TYPE "digital_inputs"
VERSION : 0.1
   STRUCT
       OtwAKPiA : Bool;    // Otawrcie szafy AKPiA
    "Czujn_Zal>0.2m" : Bool;    // Obecność w komorze AKPiA
    "Czujn_Zal>1m" : Bool;    // Obecność w komorze podziemnej
    Zasilanie : Bool;    // Obecność w komorze naziemnej
    ObcKom : Bool;    // Zalanie komory > 0.2m
    ZasilDRC : Bool;    // Zasilanie czujnika ruchu CZ1
    ZasilPompOdw : Bool;    // Zasilanie kontakorna otwarcia drzwi
    ZasilPlywZalania : Bool;    // Zasilanie czujnika ruchu CZ2
    ZasilCzujnRuchu : Bool;    // Zasilanie czujnika ruchu CZ3
    ZasilKontaktDrzwi : Bool;    // Zasilanie pływaka komory podziemnej
END_STRUCT;

END_TYPE
TYPE "digital_outputs"
VERSION : 0.1
   STRUCT
       "void" : Bool ;
   END_STRUCT;
END_TYPE
   TYPE "analog_outputs"
VERSION : 0.1
   STRUCT
       "void" : Bool ;
   END_STRUCT;
END_TYPE
   TYPE "analog_inputs"
VERSION : 0.1
   STRUCT
       FT01_Przeplyw : Int;    // Przepływ
    TTs_TempSzafy : Int;    // Temperatura szafy
    TTz_TempZewn : Int;    // Temperatura zawenętrzna
    PT07_CisnZasil_WRZ6 : Int;    // Ciśnienie w kierunku WRZ6
    PT08_CisnPowr_WRZ6 : Int;    // Ciśnienie powrotu z WRZ6
    TTk_TempKom : Int;    // Temperatura w komorze podziemnej
    PT01_CisnZasil_PLN1 : Int;    // Ciśnienie zasilania z PLN1
    PT02_CisnPowr_PLN1 : Int;    // Ciśnienie powrotu w kierunku PLN1
    PT03_CisnZasil_Bypass : Int;    // Ciśnienie zasilania Bypass
    PT04_CisnPowr_Bypass : Int;    // Ciśnienie powrotu Bypass
    PT05_CisnZasil_PLN12 : Int;    // Ciśnienie zasilania w kierunku PLN12
    PT06_CisnPowr_PLN12 : Int;    // Ciśnienie powrotu z PLN12
    TT01_TempZasil_PLN1 : Int;    // Temperatura zasliania z PLN1
    TT02_TempPowr_PLN1 : Int;    // Temperatura powrotu w kierunku PLN1
    TT04_TempPowr_WRZ6 : Int;    // Temperatura powrotu z WRZ6
    TT06_TempPowr_PLN12 : Int;    // Temperatura powrotu z PLN12
END_STRUCT;

END_TYPE

	DATA_BLOCK "DB_Input"
	VERSION : 0.1
	NON_RETAIN
	   VAR
	      inputs { S7_SetPoint := 'False'} : "digital_inputs";
	      inputs_AI : "analog_inputs";
	   END_VAR


	BEGIN

	END_DATA_BLOCK
	DATA_BLOCK "DB_Output"
	VERSION : 0.1
	NON_RETAIN
	   VAR
	      output { S7_SetPoint := 'False'} : "digital_outputs";
	      output_AO : "analog_outputs";
	   END_VAR


	BEGIN

	END_DATA_BLOCK

	FUNCTION "FC_Output" : Void
	VERSION : 0.1

	BEGIN
		"OUT" := "DB_Output".output ;
		"OUT_AO" := "DB_Output".output_AO ;
	END_FUNCTION

	FUNCTION "FC_Input" : Void
	VERSION : 0.1

	BEGIN
		"DB_Input".inputs := "IN";
		"DB_Input".inputs_AI := "IN_AI";

	END_FUNCTION
